FUNCTION_BLOCK E_D_FF_ANY (* Data latch (d) flip flop *)
  (* Standard: 61499-1 Annex A; Description: Copyright (c) 2017 fortiss GmbH, HR Agrartechnik GmbH This program and the accompanying materials are made available under the terms of the Eclipse Public License 2.0 which is available at https://www.eclipse.org/legal/epl-2.0/ SPDX-License-Identifier: EPL-2.0 *)
  (* Version 1.0, 2026-04-17, Franz H??pfinger, HR Agrartechnik GmbH, E_D_FF copied and replace BOOL by ANY *)
  PACKAGE iec61499::events;
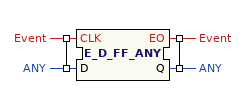
  EVENT_INPUT
    CLK WITH D; (* Clock *)
  END_EVENT
  EVENT_OUTPUT
    EO WITH Q; (* Triggered if clock results in a change of Q *)
  END_EVENT
  VAR_INPUT
    D : ANY; (* Value to latch *)
  END_VAR
  VAR_OUTPUT
    Q : ANY; (* Latched value *)
  END_VAR
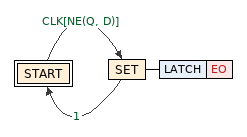
  EC_STATES
    START; (* Initial State *)
    SET : LATCH -> EO; (* Initialization *)
  END_STATES
  EC_TRANSITIONS
    SET TO START := 1;
    START TO SET := CLK[NE(Q, D)];
  END_TRANSITIONS
  ALGORITHM LATCH IN ST: (* new algorithm *)
Q := D;
  END_ALGORITHM
END_FUNCTION_BLOCK
